TYPE Type_CommOut_Drilling :
STRUCT
	s_Robot		:Type_ModuleCommOut_Drilling;
END_STRUCT
END_TYPE

(* stored: Version 1.1.0.1, ProductVersion 3.1.4024.9
   DUT Type_CommOut_Drilling: Id {c6e5e71a-dfb5-499b-aedc-e2ca5c49e947} *)
